// TIA Portal V18 export
TYPE "Console_IO_Out"
   STRUCT
      Slot4 : "DQ16x24V_Out";
      Slot5 : "AQ4xI/U_Out";
   END_STRUCT;
END_TYPE
